PROGRAM F30_PrintersCommCtrl
VAR
	fbPrinterCtrl			: ARRAY[1..cMAX_PRINTER_NUMBER] OF FB_PRINTER_DominoMSeriesCtrl;
END_VAR

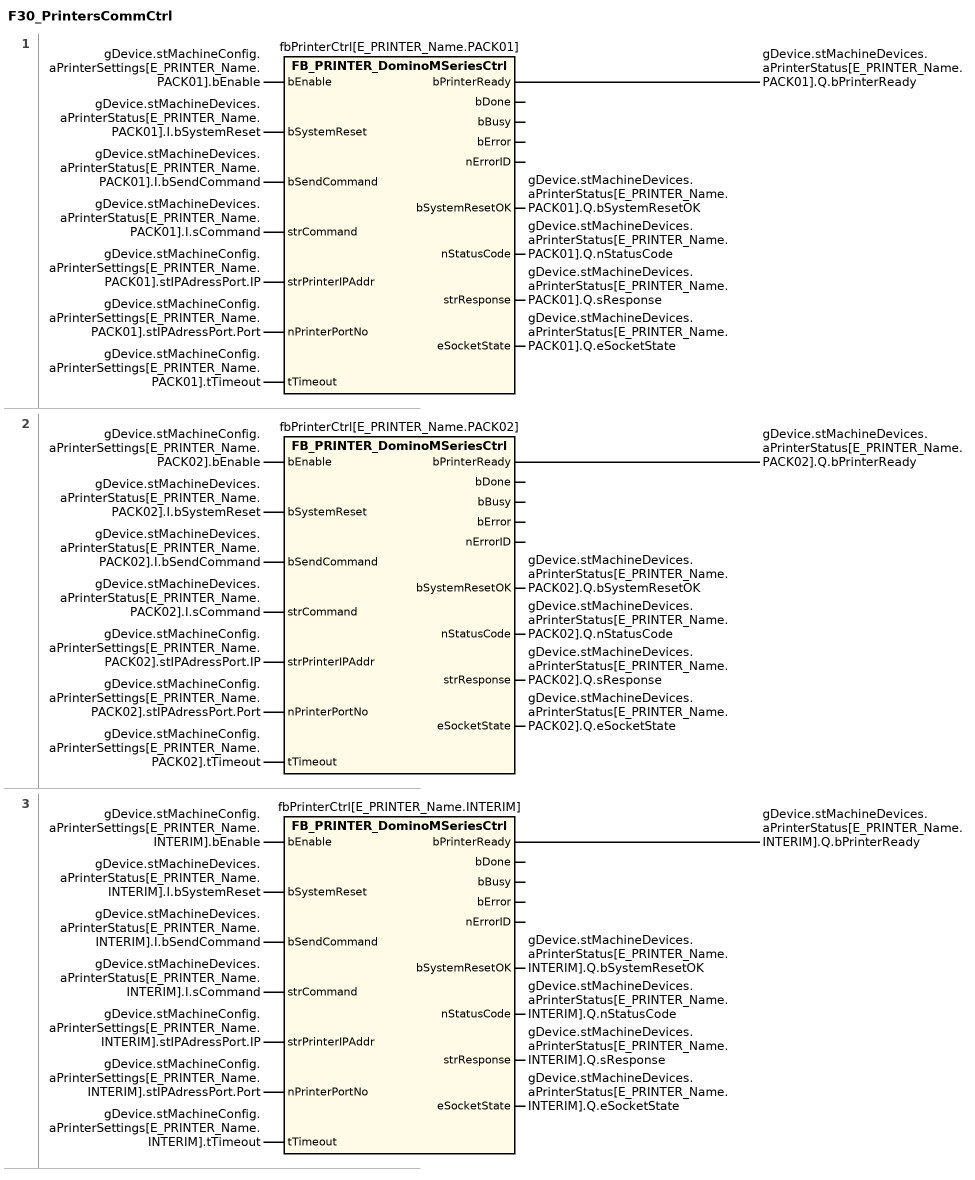
// NETWORK 1
fbPrinterCtrl[E_PRINTER_Name.PACK01](
    bEnable := gDevice.stMachineConfig.aPrinterSettings[E_PRINTER_Name.PACK01].bEnable,
    bSystemReset := gDevice.stMachineDevices.aPrinterStatus[E_PRINTER_Name.PACK01].I.bSystemReset,
    bSendCommand := gDevice.stMachineDevices.aPrinterStatus[E_PRINTER_Name.PACK01].I.bSendCommand,
    strCommand := gDevice.stMachineDevices.aPrinterStatus[E_PRINTER_Name.PACK01].I.sCommand,
    strPrinterIPAddr := gDevice.stMachineConfig.aPrinterSettings[E_PRINTER_Name.PACK01].stIPAdressPort.IP,
    nPrinterPortNo := gDevice.stMachineConfig.aPrinterSettings[E_PRINTER_Name.PACK01].stIPAdressPort.Port,
    tTimeout := gDevice.stMachineConfig.aPrinterSettings[E_PRINTER_Name.PACK01].tTimeout,
    bSystemResetOK => gDevice.stMachineDevices.aPrinterStatus[E_PRINTER_Name.PACK01].Q.bSystemResetOK,
    nStatusCode => gDevice.stMachineDevices.aPrinterStatus[E_PRINTER_Name.PACK01].Q.nStatusCode,
    strResponse => gDevice.stMachineDevices.aPrinterStatus[E_PRINTER_Name.PACK01].Q.sResponse,
    eSocketState => gDevice.stMachineDevices.aPrinterStatus[E_PRINTER_Name.PACK01].Q.eSocketState); // FB_PRINTER_DominoMSeriesCtrl
gDevice.stMachineDevices.aPrinterStatus[E_PRINTER_Name.PACK01].Q.bPrinterReady := fbPrinterCtrl[E_PRINTER_Name.PACK01].bPrinterReady;

// NETWORK 2
fbPrinterCtrl[E_PRINTER_Name.PACK02](
    bEnable := gDevice.stMachineConfig.aPrinterSettings[E_PRINTER_Name.PACK02].bEnable,
    bSystemReset := gDevice.stMachineDevices.aPrinterStatus[E_PRINTER_Name.PACK02].I.bSystemReset,
    bSendCommand := gDevice.stMachineDevices.aPrinterStatus[E_PRINTER_Name.PACK02].I.bSendCommand,
    strCommand := gDevice.stMachineDevices.aPrinterStatus[E_PRINTER_Name.PACK02].I.sCommand,
    strPrinterIPAddr := gDevice.stMachineConfig.aPrinterSettings[E_PRINTER_Name.PACK02].stIPAdressPort.IP,
    nPrinterPortNo := gDevice.stMachineConfig.aPrinterSettings[E_PRINTER_Name.PACK02].stIPAdressPort.Port,
    tTimeout := gDevice.stMachineConfig.aPrinterSettings[E_PRINTER_Name.PACK02].tTimeout,
    bSystemResetOK => gDevice.stMachineDevices.aPrinterStatus[E_PRINTER_Name.PACK02].Q.bSystemResetOK,
    nStatusCode => gDevice.stMachineDevices.aPrinterStatus[E_PRINTER_Name.PACK02].Q.nStatusCode,
    strResponse => gDevice.stMachineDevices.aPrinterStatus[E_PRINTER_Name.PACK02].Q.sResponse,
    eSocketState => gDevice.stMachineDevices.aPrinterStatus[E_PRINTER_Name.PACK02].Q.eSocketState); // FB_PRINTER_DominoMSeriesCtrl
gDevice.stMachineDevices.aPrinterStatus[E_PRINTER_Name.PACK02].Q.bPrinterReady := fbPrinterCtrl[E_PRINTER_Name.PACK02].bPrinterReady;

// NETWORK 3
fbPrinterCtrl[E_PRINTER_Name.INTERIM](
    bEnable := gDevice.stMachineConfig.aPrinterSettings[E_PRINTER_Name.INTERIM].bEnable,
    bSystemReset := gDevice.stMachineDevices.aPrinterStatus[E_PRINTER_Name.INTERIM].I.bSystemReset,
    bSendCommand := gDevice.stMachineDevices.aPrinterStatus[E_PRINTER_Name.INTERIM].I.bSendCommand,
    strCommand := gDevice.stMachineDevices.aPrinterStatus[E_PRINTER_Name.INTERIM].I.sCommand,
    strPrinterIPAddr := gDevice.stMachineConfig.aPrinterSettings[E_PRINTER_Name.INTERIM].stIPAdressPort.IP,
    nPrinterPortNo := gDevice.stMachineConfig.aPrinterSettings[E_PRINTER_Name.INTERIM].stIPAdressPort.Port,
    tTimeout := gDevice.stMachineConfig.aPrinterSettings[E_PRINTER_Name.INTERIM].tTimeout,
    bSystemResetOK => gDevice.stMachineDevices.aPrinterStatus[E_PRINTER_Name.INTERIM].Q.bSystemResetOK,
    nStatusCode => gDevice.stMachineDevices.aPrinterStatus[E_PRINTER_Name.INTERIM].Q.nStatusCode,
    strResponse => gDevice.stMachineDevices.aPrinterStatus[E_PRINTER_Name.INTERIM].Q.sResponse,
    eSocketState => gDevice.stMachineDevices.aPrinterStatus[E_PRINTER_Name.INTERIM].Q.eSocketState); // FB_PRINTER_DominoMSeriesCtrl
gDevice.stMachineDevices.aPrinterStatus[E_PRINTER_Name.INTERIM].Q.bPrinterReady := fbPrinterCtrl[E_PRINTER_Name.INTERIM].bPrinterReady;

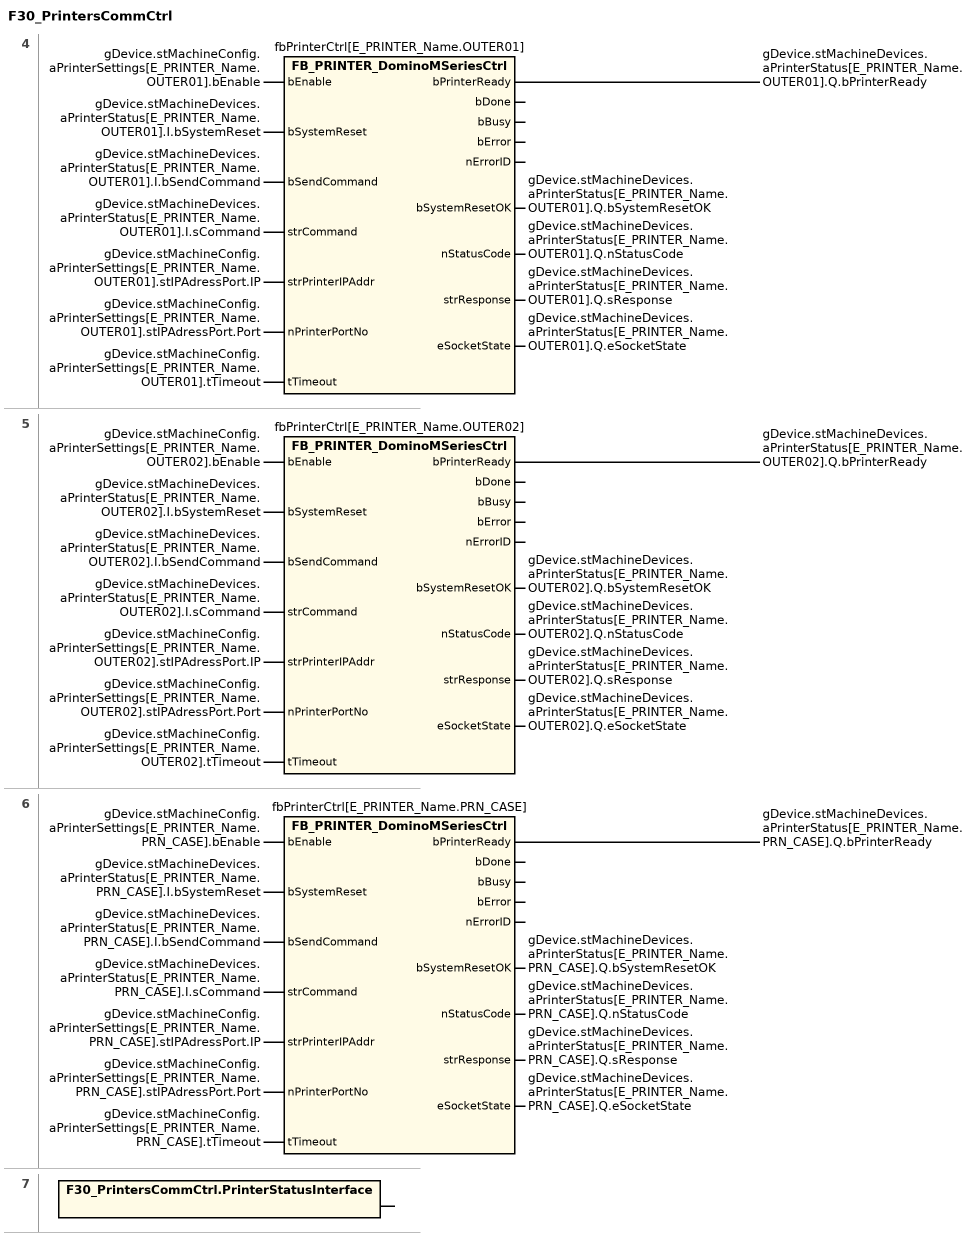
// NETWORK 4
fbPrinterCtrl[E_PRINTER_Name.OUTER01](
    bEnable := gDevice.stMachineConfig.aPrinterSettings[E_PRINTER_Name.OUTER01].bEnable,
    bSystemReset := gDevice.stMachineDevices.aPrinterStatus[E_PRINTER_Name.OUTER01].I.bSystemReset,
    bSendCommand := gDevice.stMachineDevices.aPrinterStatus[E_PRINTER_Name.OUTER01].I.bSendCommand,
    strCommand := gDevice.stMachineDevices.aPrinterStatus[E_PRINTER_Name.OUTER01].I.sCommand,
    strPrinterIPAddr := gDevice.stMachineConfig.aPrinterSettings[E_PRINTER_Name.OUTER01].stIPAdressPort.IP,
    nPrinterPortNo := gDevice.stMachineConfig.aPrinterSettings[E_PRINTER_Name.OUTER01].stIPAdressPort.Port,
    tTimeout := gDevice.stMachineConfig.aPrinterSettings[E_PRINTER_Name.OUTER01].tTimeout,
    bSystemResetOK => gDevice.stMachineDevices.aPrinterStatus[E_PRINTER_Name.OUTER01].Q.bSystemResetOK,
    nStatusCode => gDevice.stMachineDevices.aPrinterStatus[E_PRINTER_Name.OUTER01].Q.nStatusCode,
    strResponse => gDevice.stMachineDevices.aPrinterStatus[E_PRINTER_Name.OUTER01].Q.sResponse,
    eSocketState => gDevice.stMachineDevices.aPrinterStatus[E_PRINTER_Name.OUTER01].Q.eSocketState); // FB_PRINTER_DominoMSeriesCtrl
gDevice.stMachineDevices.aPrinterStatus[E_PRINTER_Name.OUTER01].Q.bPrinterReady := fbPrinterCtrl[E_PRINTER_Name.OUTER01].bPrinterReady;

// NETWORK 5
fbPrinterCtrl[E_PRINTER_Name.OUTER02](
    bEnable := gDevice.stMachineConfig.aPrinterSettings[E_PRINTER_Name.OUTER02].bEnable,
    bSystemReset := gDevice.stMachineDevices.aPrinterStatus[E_PRINTER_Name.OUTER02].I.bSystemReset,
    bSendCommand := gDevice.stMachineDevices.aPrinterStatus[E_PRINTER_Name.OUTER02].I.bSendCommand,
    strCommand := gDevice.stMachineDevices.aPrinterStatus[E_PRINTER_Name.OUTER02].I.sCommand,
    strPrinterIPAddr := gDevice.stMachineConfig.aPrinterSettings[E_PRINTER_Name.OUTER02].stIPAdressPort.IP,
    nPrinterPortNo := gDevice.stMachineConfig.aPrinterSettings[E_PRINTER_Name.OUTER02].stIPAdressPort.Port,
    tTimeout := gDevice.stMachineConfig.aPrinterSettings[E_PRINTER_Name.OUTER02].tTimeout,
    bSystemResetOK => gDevice.stMachineDevices.aPrinterStatus[E_PRINTER_Name.OUTER02].Q.bSystemResetOK,
    nStatusCode => gDevice.stMachineDevices.aPrinterStatus[E_PRINTER_Name.OUTER02].Q.nStatusCode,
    strResponse => gDevice.stMachineDevices.aPrinterStatus[E_PRINTER_Name.OUTER02].Q.sResponse,
    eSocketState => gDevice.stMachineDevices.aPrinterStatus[E_PRINTER_Name.OUTER02].Q.eSocketState); // FB_PRINTER_DominoMSeriesCtrl
gDevice.stMachineDevices.aPrinterStatus[E_PRINTER_Name.OUTER02].Q.bPrinterReady := fbPrinterCtrl[E_PRINTER_Name.OUTER02].bPrinterReady;

// NETWORK 6
fbPrinterCtrl[E_PRINTER_Name.PRN_CASE](
    bEnable := gDevice.stMachineConfig.aPrinterSettings[E_PRINTER_Name.PRN_CASE].bEnable,
    bSystemReset := gDevice.stMachineDevices.aPrinterStatus[E_PRINTER_Name.PRN_CASE].I.bSystemReset,
    bSendCommand := gDevice.stMachineDevices.aPrinterStatus[E_PRINTER_Name.PRN_CASE].I.bSendCommand,
    strCommand := gDevice.stMachineDevices.aPrinterStatus[E_PRINTER_Name.PRN_CASE].I.sCommand,
    strPrinterIPAddr := gDevice.stMachineConfig.aPrinterSettings[E_PRINTER_Name.PRN_CASE].stIPAdressPort.IP,
    nPrinterPortNo := gDevice.stMachineConfig.aPrinterSettings[E_PRINTER_Name.PRN_CASE].stIPAdressPort.Port,
    tTimeout := gDevice.stMachineConfig.aPrinterSettings[E_PRINTER_Name.PRN_CASE].tTimeout,
    bSystemResetOK => gDevice.stMachineDevices.aPrinterStatus[E_PRINTER_Name.PRN_CASE].Q.bSystemResetOK,
    nStatusCode => gDevice.stMachineDevices.aPrinterStatus[E_PRINTER_Name.PRN_CASE].Q.nStatusCode,
    strResponse => gDevice.stMachineDevices.aPrinterStatus[E_PRINTER_Name.PRN_CASE].Q.sResponse,
    eSocketState => gDevice.stMachineDevices.aPrinterStatus[E_PRINTER_Name.PRN_CASE].Q.eSocketState); // FB_PRINTER_DominoMSeriesCtrl
gDevice.stMachineDevices.aPrinterStatus[E_PRINTER_Name.PRN_CASE].Q.bPrinterReady := fbPrinterCtrl[E_PRINTER_Name.PRN_CASE].bPrinterReady;

// NETWORK 7
F30_PrintersCommCtrl.PrinterStatusInterface();

ACTION PrinterStatusInterface:
gHMI.aPrinterStatusHMI[E_PRINTER_Name.PACK01].sPrinterName :=     gDevice.stMachineConfig.aPrinterSettings[E_PRINTER_Name.PACK01].sDeviceName;
MEMMOVE(ADR(gHMI.aPrinterStatusHMI[E_PRINTER_Name.PACK01].Q), ADR(gDevice.stMachineDevices.aPrinterStatus[E_PRINTER_Name.PACK01].Q),SIZEOF(gDevice.stMachineDevices.aPrinterStatus[E_PRINTER_Name.PACK01].Q));

gHMI.aPrinterStatusHMI[E_PRINTER_Name.PACK02].sPrinterName :=     gDevice.stMachineConfig.aPrinterSettings[E_PRINTER_Name.PACK02].sDeviceName;
MEMMOVE(ADR(gHMI.aPrinterStatusHMI[E_PRINTER_Name.PACK02].Q), ADR(gDevice.stMachineDevices.aPrinterStatus[E_PRINTER_Name.PACK02].Q),SIZEOF(gDevice.stMachineDevices.aPrinterStatus[E_PRINTER_Name.PACK02].Q));

gHMI.aPrinterStatusHMI[E_PRINTER_Name.INTERIM].sPrinterName :=     gDevice.stMachineConfig.aPrinterSettings[E_PRINTER_Name.INTERIM].sDeviceName;
MEMMOVE(ADR(gHMI.aPrinterStatusHMI[E_PRINTER_Name.INTERIM].Q), ADR(gDevice.stMachineDevices.aPrinterStatus[E_PRINTER_Name.INTERIM].Q),SIZEOF(gDevice.stMachineDevices.aPrinterStatus[E_PRINTER_Name.INTERIM].Q));

gHMI.aPrinterStatusHMI[E_PRINTER_Name.OUTER01].sPrinterName :=     gDevice.stMachineConfig.aPrinterSettings[E_PRINTER_Name.OUTER01].sDeviceName;
MEMMOVE(ADR(gHMI.aPrinterStatusHMI[E_PRINTER_Name.OUTER01].Q), ADR(gDevice.stMachineDevices.aPrinterStatus[E_PRINTER_Name.OUTER01].Q),SIZEOF(gDevice.stMachineDevices.aPrinterStatus[E_PRINTER_Name.OUTER01].Q));

gHMI.aPrinterStatusHMI[E_PRINTER_Name.OUTER02].sPrinterName :=     gDevice.stMachineConfig.aPrinterSettings[E_PRINTER_Name.OUTER02].sDeviceName;
MEMMOVE(ADR(gHMI.aPrinterStatusHMI[E_PRINTER_Name.OUTER02].Q), ADR(gDevice.stMachineDevices.aPrinterStatus[E_PRINTER_Name.OUTER02].Q),SIZEOF(gDevice.stMachineDevices.aPrinterStatus[E_PRINTER_Name.OUTER02].Q));

gHMI.aPrinterStatusHMI[E_PRINTER_Name.PRN_CASE].sPrinterName :=     gDevice.stMachineConfig.aPrinterSettings[E_PRINTER_Name.PRN_CASE].sDeviceName;
MEMMOVE(ADR(gHMI.aPrinterStatusHMI[E_PRINTER_Name.PRN_CASE].Q), ADR(gDevice.stMachineDevices.aPrinterStatus[E_PRINTER_Name.PRN_CASE].Q),SIZEOF(gDevice.stMachineDevices.aPrinterStatus[E_PRINTER_Name.PRN_CASE].Q));
END_ACTION

END_PROGRAM

(* stored: Version 1.1.0.1
   POU F30_PrintersCommCtrl: Id {f095d8f3-19b9-449f-adcc-3c85c45b4de6}, SpecialFunc None
   Action PrinterStatusInterface: Id {090cc5e7-ede9-40d2-bbb4-d8df2b4a9527} *)
